Universal Robots PolyScope program: networking_xmlrpc_client.urp

Program rpc_client (createdIn=3.4.5.100 lastSavedIn=3.4.5.100 directory=/programs/usbdisk installation=default robotSerialNumber=2016353011)
Calibrated DH parameters: a=[0.000233, -0.180339, -0.373678, -0.000024, 0.000135, 0]; d=[0.089179, 873.064081, -854.282843, -18.670907, 0.09475, 0.082522]; alpha=[1.570027, -0.00044, -0.006312, 1.570545, -1.570879, 0]; deltaTheta=[-0.000037, -1.132248, 0.825087, 0.307217, 0.000011, 0.000228]
Robot Program (runOnlyOnce=false motionType=MoveJ speed=1.047198 acceleration=1.396263 useActiveTCP=false)
  Script: gripper = rpc_factory("xmlrpc","http://10.1.12.85:8008/RPC2")
  Script: gripper.close_gripper()
  Script: gripper.open_gripper()
  Script: gripper.set_gripper_torque(50)
  var_1 := gripper.get_target_pose()
  MoveJ speed 60 deg/s, acceleration 80 deg/s^2 (useActiveTCP=true)
    Waypoint Waypoint_1 (Variable): variable=var_1
